// TIA Portal V18 export
FUNCTION "settShiftParTransfer" : Void   // FC5, FBD
{ S7_Optimized_Access := 'TRUE' }
// stored: SetENOAutomatically false
   VAR_INPUT
      settShiftParEN : DInt;
      settShiftParVal : DInt;
   END_VAR
   VAR_IN_OUT
      settingsParameter : DInt;
   END_VAR
BEGIN

REGION Network 1
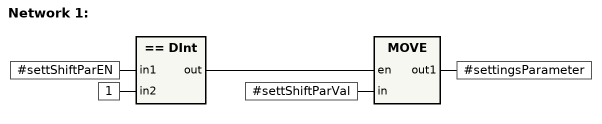
   IF #settShiftParEN = 1 THEN #settingsParameter := #settShiftParVal; END_IF;
END_REGION
END_FUNCTION
